(* CoDeSys 2.3.9.50 project: 6D.pr6 *)
(* Libraries: STANDARD.LB6 5.6.98 12:03:02 *)

(* POU MAIN, LD *)
PROGRAM MAIN
VAR
	Start AT %IX0.0: BOOL;
	T1: TOF;
	increase5 AT %QX0.0: BOOL;
	decrease5 AT %QX0.1: BOOL;
	Increasetime AT %IX0.1: BOOL;
	DecreaseTime AT %IX0.2: BOOL;
	timechange: TIME := t#5s;
	A AT %QX0.2: BOOL;
	B AT %QX0.3: BOOL;
END_VAR
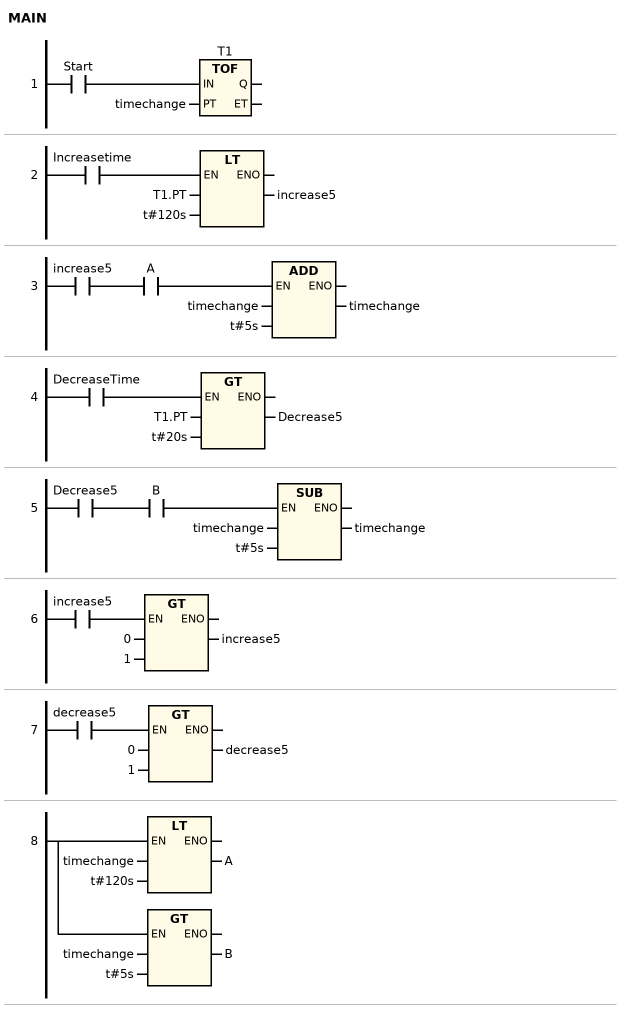
_LD_ (* Ladder Diagram *)
NETWORK 1
	[Start] - T1:TOF(IN: *, PT: timechange)
NETWORK 2
	[Increasetime]
		EN --- LT(T1.PT, t#120s) => increase5
NETWORK 3
	[increase5] - [A]
		EN --- ADD(timechange, t#5s) => timechange
NETWORK 4
	[DecreaseTime]
		EN --- GT(T1.PT, t#20s) => Decrease5
NETWORK 5
	[Decrease5] - [B]
		EN --- SUB(timechange, t#5s) => timechange
NETWORK 6
	[increase5]
		EN --- GT(0, 1) => increase5
NETWORK 7
	[decrease5]
		EN --- GT(0, 1) => decrease5
NETWORK 8
	*
		EN --- LT(timechange, t#120s) => A
		EN --- GT(timechange, t#5s) => B
_END_LD_
(* the same logic as Structured Text *)
(* Network 1 *)
T1(IN := Start, PT := timechange);
(* Network 2 *)
IF Increasetime THEN
	increase5 := T1.PT < t#120s;
END_IF;
(* Network 3 *)
IF increase5 AND A THEN
	timechange := timechange + t#5s;
END_IF;
(* Network 4 *)
IF DecreaseTime THEN
	Decrease5 := T1.PT > t#20s;
END_IF;
(* Network 5 *)
IF Decrease5 AND B THEN
	timechange := timechange - t#5s;
END_IF;
(* Network 6 *)
IF increase5 THEN
	increase5 := 0 > 1;
END_IF;
(* Network 7 *)
IF decrease5 THEN
	decrease5 := 0 > 1;
END_IF;
(* Network 8 *)
A := timechange < t#120s;
B := timechange > t#5s;
END_PROGRAM
